// TIA Portal V18 export
// export: Created 2026-01-09T11:31:56.0663809Z, ExportSetting WithDefaults, DisplayName Totally Integrated Automation Portal, DisplayVersion V18 Update 5, DisplayName TIA Portal Openness, DisplayVersion V18 Update 5, DisplayName TIA Portal Teamcenter Gateway, DisplayVersion V18, DisplayName TIA Portal Version Control Interface, DisplayVersion V18, DisplayName SINAMICS Startdrive Advanced, DisplayVersion V18 SP2 Update 1, DisplayName SINAMICS Startdrive G110M, G120, G120C, G120D, G120P, G115D, DisplayVersion V18 SP2 Update 1, DisplayName SINAMICS Startdrive G130, G150, S120, S150, SINAMICS MV, S210, G220, S200, DisplayVersion V18 SP2 Update 1, DisplayName STEP 7 Professional, DisplayVersion V18 Update 5, DisplayName STEP 7 Safety, DisplayVersion V18, DisplayName WinCC Professional, DisplayVersion V18 Update 5
TagTable "ST350_SafetyGate"
  ST10_SafetyGate_InterfaceDB_aDev{1} : SafetyGateUDT  (PLC tag ST10_SafetyGate_InterfaceDB.aDev[1], CPU S71500-2PN_TP700, 100 ms)
    TagStructureMember "CMD"
      TagStructureMember "RequestPB"
    TagStructureMember "Status"
      TagStructureMember "Lock/Unlock Indicator"
      TagStructureMember "INT"
      TagStructureMember "Locked"
      TagStructureMember "Unlocked"
      TagStructureMember "Opened"
  ST10_SafetyGate_InterfaceDB_aDev{2} : SafetyGateUDT  (PLC tag ST10_SafetyGate_InterfaceDB.aDev[2], CPU S71500-2PN_TP700, 100 ms)
    TagStructureMember "CMD"
      TagStructureMember "RequestPB"
    TagStructureMember "Status"
      TagStructureMember "Lock/Unlock Indicator"
      TagStructureMember "INT"
      TagStructureMember "Locked"
      TagStructureMember "Unlocked"
      TagStructureMember "Opened"
  ST10_SafetyGate_InterfaceDB_aDev{3} : SafetyGateUDT  (PLC tag ST10_SafetyGate_InterfaceDB.aDev[3], CPU S71500-2PN_TP700, 100 ms)
    TagStructureMember "CMD"
      TagStructureMember "RequestPB"
    TagStructureMember "Status"
      TagStructureMember "Lock/Unlock Indicator"
      TagStructureMember "INT"
      TagStructureMember "Locked"
      TagStructureMember "Unlocked"
      TagStructureMember "Opened"
  ST10_SafetyGate_InterfaceDB_aDev{4} : SafetyGateUDT  (PLC tag ST10_SafetyGate_InterfaceDB.aDev[4], CPU S71500-2PN_TP700, 100 ms)
    TagStructureMember "CMD"
      TagStructureMember "RequestPB"
    TagStructureMember "Status"
      TagStructureMember "Lock/Unlock Indicator"
      TagStructureMember "INT"
      TagStructureMember "Locked"
      TagStructureMember "Unlocked"
      TagStructureMember "Opened"
  ST10_SafetyGate_InterfaceDB_aDev{5} : SafetyGateUDT  (PLC tag ST10_SafetyGate_InterfaceDB.aDev[5], CPU S71500-2PN_TP700, 100 ms)
    TagStructureMember "CMD"
      TagStructureMember "RequestPB"
    TagStructureMember "Status"
      TagStructureMember "Lock/Unlock Indicator"
      TagStructureMember "INT"
      TagStructureMember "Locked"
      TagStructureMember "Unlocked"
      TagStructureMember "Opened"
  ST10_SafetyGate_InterfaceDB_aDev{7} : SafetyGateUDT  (PLC tag ST10_SafetyGate_InterfaceDB.aDev[7], CPU S71500-2PN_TP700, 100 ms)
    TagStructureMember "CMD"
      TagStructureMember "RequestPB"
    TagStructureMember "Status"
      TagStructureMember "Lock/Unlock Indicator"
      TagStructureMember "INT"
      TagStructureMember "Locked"
      TagStructureMember "Unlocked"
      TagStructureMember "Opened"
  ST10_SafetyGate_InterfaceDB_aDev{8} : SafetyGateUDT  (PLC tag ST10_SafetyGate_InterfaceDB.aDev[8], CPU S71500-2PN_TP700, 100 ms)
    TagStructureMember "CMD"
      TagStructureMember "RequestPB"
    TagStructureMember "Status"
      TagStructureMember "Lock/Unlock Indicator"
      TagStructureMember "INT"
      TagStructureMember "Locked"
      TagStructureMember "Unlocked"
      TagStructureMember "Opened"
  ST10_SafetyGate_InterfaceDB_aDev{9} : SafetyGateUDT  (PLC tag ST10_SafetyGate_InterfaceDB.aDev[9], CPU S71500-2PN_TP700, 100 ms)
    TagStructureMember "CMD"
      TagStructureMember "RequestPB"
    TagStructureMember "Status"
      TagStructureMember "Lock/Unlock Indicator"
      TagStructureMember "INT"
      TagStructureMember "Locked"
      TagStructureMember "Unlocked"
      TagStructureMember "Opened"
  ST10_SafetyGate_InterfaceDB_aDev{10} : SafetyGateUDT  (PLC tag ST10_SafetyGate_InterfaceDB.aDev[10], CPU S71500-2PN_TP700, 100 ms)
    TagStructureMember "CMD"
      TagStructureMember "RequestPB"
    TagStructureMember "Status"
      TagStructureMember "Lock/Unlock Indicator"
      TagStructureMember "INT"
      TagStructureMember "Locked"
      TagStructureMember "Unlocked"
      TagStructureMember "Opened"
  ST10_SafetyGate_InterfaceDB_aDev{11} : SafetyGateUDT  (PLC tag ST10_SafetyGate_InterfaceDB.aDev[11], CPU S71500-2PN_TP700, 100 ms)
    TagStructureMember "CMD"
      TagStructureMember "RequestPB"
    TagStructureMember "Status"
      TagStructureMember "Lock/Unlock Indicator"
      TagStructureMember "INT"
      TagStructureMember "Locked"
      TagStructureMember "Unlocked"
      TagStructureMember "Opened"
  ST10_SafetyGate_InterfaceDB_aDev{12} : SafetyGateUDT  (PLC tag ST10_SafetyGate_InterfaceDB.aDev[12], CPU S71500-2PN_TP700, 100 ms)
    TagStructureMember "CMD"
      TagStructureMember "RequestPB"
    TagStructureMember "Status"
      TagStructureMember "Lock/Unlock Indicator"
      TagStructureMember "INT"
      TagStructureMember "Locked"
      TagStructureMember "Unlocked"
      TagStructureMember "Opened"
  ST10_SafetyGate_InterfaceDB_aDev{13} : SafetyGateUDT  (PLC tag ST10_SafetyGate_InterfaceDB.aDev[13], CPU S71500-2PN_TP700, 100 ms)
    TagStructureMember "CMD"
      TagStructureMember "RequestPB"
    TagStructureMember "Status"
      TagStructureMember "Lock/Unlock Indicator"
      TagStructureMember "INT"
      TagStructureMember "Locked"
      TagStructureMember "Unlocked"
      TagStructureMember "Opened"
  ST10_SafetyGate_InterfaceDB_aDev{14} : SafetyGateUDT  (PLC tag ST10_SafetyGate_InterfaceDB.aDev[14], CPU S71500-2PN_TP700, 100 ms)
    TagStructureMember "CMD"
      TagStructureMember "RequestPB"
    TagStructureMember "Status"
      TagStructureMember "Lock/Unlock Indicator"
      TagStructureMember "INT"
      TagStructureMember "Locked"
      TagStructureMember "Unlocked"
      TagStructureMember "Opened"
  ST10_SafetyGate_InterfaceDB_aDev{15} : SafetyGateUDT  (PLC tag ST10_SafetyGate_InterfaceDB.aDev[15], CPU S71500-2PN_TP700, 100 ms)
    TagStructureMember "CMD"
      TagStructureMember "RequestPB"
    TagStructureMember "Status"
      TagStructureMember "Lock/Unlock Indicator"
      TagStructureMember "INT"
      TagStructureMember "Locked"
      TagStructureMember "Unlocked"
      TagStructureMember "Opened"
  ST10_SafetyGate_InterfaceDB_aDev{16} : SafetyGateUDT  (PLC tag ST10_SafetyGate_InterfaceDB.aDev[16], CPU S71500-2PN_TP700, 100 ms)
    TagStructureMember "CMD"
      TagStructureMember "RequestPB"
    TagStructureMember "Status"
      TagStructureMember "Lock/Unlock Indicator"
      TagStructureMember "INT"
      TagStructureMember "Locked"
      TagStructureMember "Unlocked"
      TagStructureMember "Opened"
  ST10_SafetyGate_InterfaceDB_aDev{17} : SafetyGateUDT  (PLC tag ST10_SafetyGate_InterfaceDB.aDev[17], CPU S71500-2PN_TP700, 100 ms)
    TagStructureMember "CMD"
      TagStructureMember "RequestPB"
    TagStructureMember "Status"
      TagStructureMember "Lock/Unlock Indicator"
      TagStructureMember "INT"
      TagStructureMember "Locked"
      TagStructureMember "Unlocked"
      TagStructureMember "Opened"
  ST10_SafetyGate_InterfaceDB_aDev{18} : SafetyGateUDT  (PLC tag ST10_SafetyGate_InterfaceDB.aDev[18], CPU S71500-2PN_TP700, 100 ms)
    TagStructureMember "CMD"
      TagStructureMember "RequestPB"
    TagStructureMember "Status"
      TagStructureMember "Lock/Unlock Indicator"
      TagStructureMember "INT"
      TagStructureMember "Locked"
      TagStructureMember "Unlocked"
      TagStructureMember "Opened"
  ST10_SafetyGate_InterfaceDB_aDev{19} : SafetyGateUDT  (PLC tag ST10_SafetyGate_InterfaceDB.aDev[19], CPU S71500-2PN_TP700, 100 ms)
    TagStructureMember "CMD"
      TagStructureMember "RequestPB"
    TagStructureMember "Status"
      TagStructureMember "Lock/Unlock Indicator"
      TagStructureMember "INT"
      TagStructureMember "Locked"
      TagStructureMember "Unlocked"
      TagStructureMember "Opened"
  ST10_SafetyGate_InterfaceDB_aDev{20} : SafetyGateUDT  (PLC tag ST10_SafetyGate_InterfaceDB.aDev[20], CPU S71500-2PN_TP700, 100 ms)
    TagStructureMember "CMD"
      TagStructureMember "RequestPB"
    TagStructureMember "Status"
      TagStructureMember "Lock/Unlock Indicator"
      TagStructureMember "INT"
      TagStructureMember "Locked"
      TagStructureMember "Unlocked"
      TagStructureMember "Opened"
  ST10_SafetyGate_InterfaceDB_aDev{6} : SafetyGateUDT  (PLC tag ST10_SafetyGate_InterfaceDB.aDev[6], CPU S71500-2PN_TP700, 100 ms)
    TagStructureMember "CMD"
      TagStructureMember "RequestPB"
    TagStructureMember "Status"
      TagStructureMember "Lock/Unlock Indicator"
      TagStructureMember "INT"
      TagStructureMember "Locked"
      TagStructureMember "Unlocked"
      TagStructureMember "Opened"
